// TIA Portal project "Prakticne-5" (V16)

(* hardware
DEVICE "S7-1200 station_1"  S7-1200 Station
   slot 0: "Rack_0"  S7-1200 Rack  Rack  V1.0
   slot 1: "PLC_1"  CPU 1214C AC/DC/Rly  6ES7 214-1BG31-0XB0  V3.0
*)

// ===== PLC "PLC_1"  CPU 1214C AC/DC/Rly =====

VAR_GLOBAL   // PLC tag table "Default tag table"
   "Clock_Byte" AT %MB10 : Byte;
   "Clock_10Hz" AT %M10.0 : Bool;
   "Clock_5Hz" AT %M10.1 : Bool;
   "Clock_2.5Hz" AT %M10.2 : Bool;
   "Clock_2Hz" AT %M10.3 : Bool;
   "Clock_1.25Hz" AT %M10.4 : Bool;
   "Clock_1Hz" AT %M10.5 : Bool;
   "Clock_0.625Hz" AT %M10.6 : Bool;
   "Clock_0.5Hz" AT %M10.7 : Bool;
   "Tag_1" AT %M30.0 : Bool;
   "Tag_2" AT %M40.0 : Bool;
   "Tag_3" AT %M40.2 : Bool;
   "Tag_4" AT %M50.0 : Bool;
   "Tag_5" AT %M45.0 : Bool;
   "Tag_6" AT %M60.0 : Bool;
   "Tag_7" AT %M100.1 : Bool;
   "Tag_8" AT %M100.2 : Bool;
   "Tag_9" AT %M110.3 : Bool;
   "Tag_10" AT %M120.0 : Bool;
END_VAR

VAR_GLOBAL   // PLC tag table "Tag table_1"
   "Prekidac 1" AT %I0.0 : Bool;
   "Prekidac 2" AT %I0.1 : Bool;
   "Prekidac 3" AT %I0.2 : Bool;
   "Prekidac 4" AT %I0.3 : Bool;
   "Prekidac 5" AT %I0.4 : Bool;
   "Prekidac 6" AT %I0.5 : Bool;
   "Prekidac 7" AT %I0.6 : Bool;
   "Induktivni senzor" AT %I1.0 : Bool;
   "Pun krig napravljen" AT %I1.1 : Bool;
   "Dioda 2" AT %Q0.0 : Bool;
   "Dioda 3" AT %Q0.1 : Bool;
   "Dioda 4" AT %Q0.2 : Bool;
   "Dioda 5" AT %Q0.3 : Bool;
   "Motor suprotno od kazaljke" AT %Q0.4 : Bool;
   "Motor u smeru kazaljke" AT %Q0.5 : Bool;
END_VAR

// folder: System blocks/Program resources

DATA_BLOCK "Brojac_cw"   // DB1
{ S7_Optimized_Access := 'TRUE' }
AUTHOR : Simatic
FAMILY : IEC
NAME : CNTR
VERSION : 1.0
// stored: InstanceOfName IEC_COUNTER
"IEC_COUNTER"
BEGIN
END_DATA_BLOCK

DATA_BLOCK "10s_medju_pauza"   // DB2
{ S7_Optimized_Access := 'TRUE' }
AUTHOR : Simatic
FAMILY : IEC
NAME : IEC_TMR
VERSION : 1.0
// stored: InstanceOfName IEC_TIMER
"IEC_TIMER"
BEGIN
END_DATA_BLOCK

DATA_BLOCK "Brojac_ccw"   // DB3
{ S7_Optimized_Access := 'TRUE' }
AUTHOR : Simatic
FAMILY : IEC
NAME : CNTR
VERSION : 1.0
// stored: InstanceOfName IEC_COUNTER
"IEC_COUNTER"
BEGIN
END_DATA_BLOCK

DATA_BLOCK "Timer_on"   // DB5
{ S7_Optimized_Access := 'TRUE' }
AUTHOR : Simatic
FAMILY : IEC
NAME : IEC_TMR
VERSION : 1.0
// stored: InstanceOfName IEC_TIMER
"IEC_TIMER"
BEGIN
END_DATA_BLOCK

// folder: (top level)

FUNCTION "FC_kretanje" : Void   // FC1, LAD
{ S7_Optimized_Access := 'TRUE' }
VERSION : 0.1
   VAR_TEMP   // added for the SCL form of the ladder/FBD networks
      _w1 : Bool;
   END_VAR
BEGIN

REGION Network 1
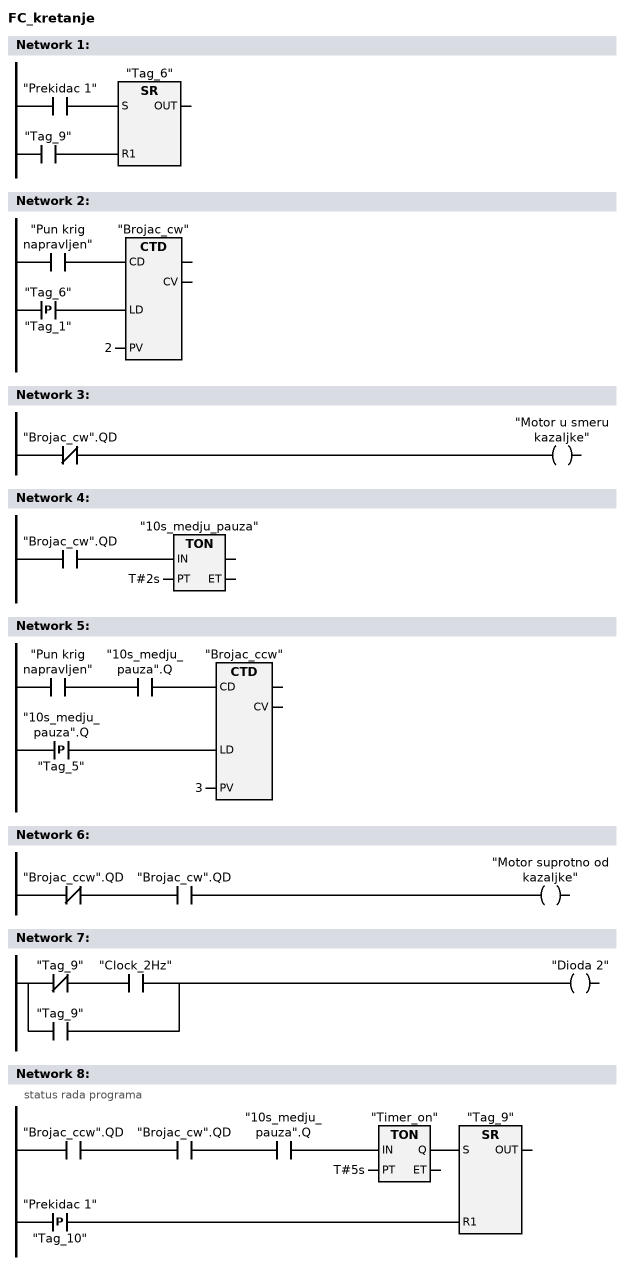
   RUNG wire#powerrail
      Contact( "Prekidac 1" )
      S_SR(operand := "Tag_6", r1 := wire#w1)
   END_RUNG
   RUNG wire#powerrail
      Contact( "Tag_9" )
   END_RUNG wire#w1
   // the same network as SCL:
   IF "Prekidac 1" THEN
       "Tag_6" := TRUE;   // SR flip-flop
   END_IF;
   IF "Tag_9" THEN "Tag_6" := FALSE; END_IF;
END_REGION

REGION Network 2
   #_w1 := "Tag_6" AND NOT "Tag_1";   // rising edge of "Tag_6"
   "Tag_1" := "Tag_6";
   "Brojac_cw".CTD(CD := "Pun krig napravljen", LD := #_w1, PV := 2);
END_REGION

REGION Network 3
   RUNG wire#powerrail
      I_Contact( "Brojac_cw".QD )
      Coil( "Motor u smeru kazaljke" )
   END_RUNG
   // the same network as SCL:
   "Motor u smeru kazaljke" := NOT "Brojac_cw".QD;
END_REGION

REGION Network 4
   "10s_medju_pauza".TON(IN := "Brojac_cw".QD, PT := T#2s);
END_REGION

REGION Network 5
   #_w1 := "10s_medju_pauza".Q AND NOT "Tag_5";   // rising edge of "10s_medju_pauza".Q
   "Tag_5" := "10s_medju_pauza".Q;
   "Brojac_ccw".CTD(CD := "Pun krig napravljen" AND "10s_medju_pauza".Q, LD := #_w1, PV := 3);
END_REGION

REGION Network 6
   RUNG wire#powerrail
      I_Contact( "Brojac_ccw".QD )
      Contact( "Brojac_cw".QD )
      Coil( "Motor suprotno od kazaljke" )
   END_RUNG
   // the same network as SCL:
   "Motor suprotno od kazaljke" := NOT "Brojac_ccw".QD AND "Brojac_cw".QD;
END_REGION

REGION Network 7
   RUNG wire#powerrail
      I_Contact( "Tag_9" )
      Contact( "Clock_2Hz" )
      wire#w1
      Coil( "Dioda 2" )
   END_RUNG
   RUNG wire#powerrail
      Contact( "Tag_9" )
   END_RUNG wire#w1
   // the same network as SCL:
   "Dioda 2" := (NOT "Tag_9" AND "Clock_2Hz") OR "Tag_9";
END_REGION

REGION Network 8
   // status rada programa
   "Timer_on".TON(IN := "Brojac_ccw".QD AND "Brojac_cw".QD AND "10s_medju_pauza".Q, PT := T#5s);
   #_w1 := "Prekidac 1" AND NOT "Tag_10";   // rising edge of "Prekidac 1"
   "Tag_10" := "Prekidac 1";
   IF "Timer_on".Q THEN
       "Tag_9" := TRUE;   // SR flip-flop
   END_IF;
   IF #_w1 THEN "Tag_9" := FALSE; END_IF;
END_REGION
END_FUNCTION

ORGANIZATION_BLOCK "Main"   // OB1, LAD, ProgramCycle
TITLE = "Main Program Sweep (Cycle)"
{ S7_Optimized_Access := 'TRUE' }
VERSION : 0.1
BEGIN

REGION Network 1
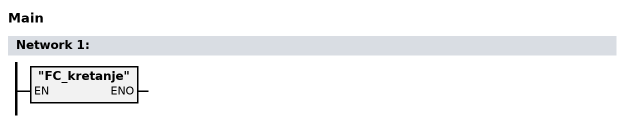
   RUNG wire#powerrail
      "FC_kretanje"()
   END_RUNG
   // the same network as SCL:
   "FC_kretanje"();
END_REGION
END_ORGANIZATION_BLOCK